// TIA Portal V20 export
TYPE "typeScrapBoxMonitoring"
// stored: Access Published, IsFailsafeCompliant true, Namespace Safety
   STRUCT
      lock : Bool;   // Scrap Box Locked Signal
      unlock : Bool;   // Scrap Box UnLocked Signal
      reset : Bool;   // Scrap Box Reset Signal
      error : Bool;   // Scrap Box Error Signal
   END_STRUCT;
END_TYPE
